// TIA Portal V20 export
TYPE "LER_typeServoTorqueCalMonitoring"
// stored: Access Published
   STRUCT
      OverLoad_Warning : Bool;
      OverLoad_Alarm : Bool;
      OverLoad_Warning_SV : LReal;
      OverLoad_Alarm_SV : LReal;
      Actual_Torque : LReal;
      Average_Torque : LReal;
      Peak_Torque : LReal;
      Current_load : LReal;
      Average_load : LReal;
      Peak_load : LReal;
   END_STRUCT;
END_TYPE
